{attribute 'OPC.UA.DA' := '1'}
{attribute 'analysis' := '-33'}
TYPE DUT_TestStruct2 :
STRUCT
	ByteValue			:BYTE			:= 16#FF;
	WordValue			:WORD			:= 16#FFFF;
	DWordValue			:DWORD			:= 16#FFFF_FFFF;
	LWordValue			:LWORD			:= 16#FFFF_FFFF_FFFF_FFFF;
END_STRUCT
END_TYPE

(* stored: Version 1.1.0.1, ProductVersion 3.1.4024.9
   DUT DUT_TestStruct2: Id {3b1a7687-6a60-4de7-859c-f4e40aa65cf7} *)
